(* IEC 61131-3 sources: festo-codesys-mcp/knowledge/library/sensors, 4 files *)

(* ---- FB_AnalogInput.st ---- *)
(* =============================================================
   FB_AnalogInput — Generic Analog Input with Scaling and Filtering

   Category:     Sensors
   Platform:     CODESYS V3.5 (IEC 61131-3)
   Version:      1.0
   Dependencies: None (standard IEC only)

   General-purpose analog input block with linear scaling from
   raw ADC to engineering units, first-order filtering, and
   high/low alarm limits.

   Usage:
     fbPressure : FB_AnalogInput;
     fbPressure(nRawValue := nAD_Ch1,
                rScaleMin := 0.0, rScaleMax := 10.0,
                sUnit := 'bar');
     rPressure := fbPressure.rValue;
   ============================================================= *)
FUNCTION_BLOCK FB_AnalogInput
VAR_INPUT
    nRawValue       : INT;                 (* Raw ADC value *)
    rScaleMin       : REAL := 0.0;         (* Engineering minimum *)
    rScaleMax       : REAL := 100.0;       (* Engineering maximum *)
    nRawMin         : INT := 0;            (* ADC raw minimum *)
    nRawMax         : INT := 32767;        (* ADC raw maximum *)
    rAlarmHigh      : REAL := 90.0;        (* High alarm limit *)
    rAlarmLow       : REAL := 5.0;         (* Low alarm limit *)
    rHysteresis     : REAL := 2.0;         (* Alarm hysteresis *)
    rFilterFactor   : REAL := 0.2;         (* Filter alpha (0.0-1.0) *)
    bEnable         : BOOL := TRUE;        (* Enable processing *)
END_VAR
VAR_OUTPUT
    rValue          : REAL;                (* Scaled value *)
    rPercent        : REAL;                (* 0-100% of scale *)
    bAlarmHigh      : BOOL;                (* High alarm *)
    bAlarmLow       : BOOL;                (* Low alarm *)
    bValid          : BOOL;                (* Reading valid *)
END_VAR
VAR
    rFiltered       : REAL;
    rRange          : REAL;
    bInit           : BOOL := FALSE;
END_VAR

IF NOT bEnable THEN
    bValid := FALSE;
    RETURN;
END_IF

(* Filter *)
IF NOT bInit THEN
    rFiltered := INT_TO_REAL(nRawValue);
    bInit := TRUE;
ELSE
    rFiltered := rFiltered + rFilterFactor * (INT_TO_REAL(nRawValue) - rFiltered);
END_IF

(* Scale *)
rRange := INT_TO_REAL(nRawMax - nRawMin);
IF ABS(rRange) > 0.001 THEN
    rValue := (rFiltered - INT_TO_REAL(nRawMin)) / rRange
              * (rScaleMax - rScaleMin) + rScaleMin;
    rPercent := (rFiltered - INT_TO_REAL(nRawMin)) / rRange * 100.0;
ELSE
    rValue := rScaleMin;
    rPercent := 0.0;
END_IF
bValid := TRUE;

(* Alarms with hysteresis *)
IF rValue >= rAlarmHigh THEN
    bAlarmHigh := TRUE;
ELSIF rValue < (rAlarmHigh - rHysteresis) THEN
    bAlarmHigh := FALSE;
END_IF

IF rValue <= rAlarmLow THEN
    bAlarmLow := TRUE;
ELSIF rValue > (rAlarmLow + rHysteresis) THEN
    bAlarmLow := FALSE;
END_IF

END_FUNCTION_BLOCK

(* ---- FB_FlowSensor.st ---- *)
(* =============================================================
   FB_FlowSensor — Flow Rate Sensor with Totalization

   Category:     Sensors
   Platform:     CODESYS V3.5 (IEC 61131-3)
   Version:      1.0
   Dependencies: None (standard IEC only)

   Monitors flow rate from analog sensor (4-20mA/0-10V).
   Includes low-flow alarm, totalization (accumulated volume),
   and peak flow tracking.

   Usage:
     fbFlow : FB_FlowSensor;
     fbFlow(nRawValue := nAD_Flow,
            rScaleMin := 0.0, rScaleMax := 50.0,
            rAlarmLow := 5.0, tCycleTime := T#100MS);
     rFlowRate  := fbFlow.rValue;
     rTotalVol  := fbFlow.rTotalVolume;
     bNoFlow    := fbFlow.bAlarmLow;
   ============================================================= *)
FUNCTION_BLOCK FB_FlowSensor
VAR_INPUT
    nRawValue       : INT;                 (* Raw ADC value *)
    rScaleMin       : REAL := 0.0;         (* Flow min [L/min] *)
    rScaleMax       : REAL := 50.0;        (* Flow max [L/min] *)
    nRawMin         : INT := 0;            (* ADC minimum *)
    nRawMax         : INT := 32767;        (* ADC maximum *)
    rAlarmLow       : REAL := 5.0;         (* Low flow alarm [L/min] *)
    rHysteresis     : REAL := 1.0;         (* Alarm hysteresis *)
    rFilterFactor   : REAL := 0.15;        (* Filter alpha *)
    tCycleTime      : TIME := T#100MS;     (* PLC scan cycle *)
    bEnable         : BOOL := TRUE;        (* Enable sensor *)
    bResetTotal     : BOOL;                (* Reset totalizer *)
END_VAR
VAR_OUTPUT
    rValue          : REAL;                (* Flow rate [L/min] *)
    rTotalVolume    : REAL := 0.0;         (* Accumulated volume [L] *)
    rPeakFlow       : REAL := 0.0;         (* Peak flow recorded *)
    bAlarmLow       : BOOL;                (* Low flow alarm *)
    bNoFlow         : BOOL;                (* Zero flow detected *)
    bValid          : BOOL;                (* Reading valid *)
END_VAR
VAR
    rFiltered       : REAL;
    rRange          : REAL;
    rDtMin          : REAL;
    bInit           : BOOL := FALSE;
END_VAR

IF bResetTotal THEN
    rTotalVolume := 0.0;
    rPeakFlow := 0.0;
END_IF

IF NOT bEnable THEN
    bValid := FALSE;
    RETURN;
END_IF

(* Filter *)
IF NOT bInit THEN
    rFiltered := INT_TO_REAL(nRawValue);
    bInit := TRUE;
ELSE
    rFiltered := rFiltered + rFilterFactor * (INT_TO_REAL(nRawValue) - rFiltered);
END_IF

(* Scale *)
rRange := INT_TO_REAL(nRawMax - nRawMin);
IF ABS(rRange) > 0.001 THEN
    rValue := (rFiltered - INT_TO_REAL(nRawMin)) / rRange
              * (rScaleMax - rScaleMin) + rScaleMin;
ELSE
    rValue := 0.0;
END_IF
IF rValue < 0.0 THEN rValue := 0.0; END_IF
bValid := TRUE;

(* Totalization: flow [L/min] * dt [min] = volume [L] *)
rDtMin := TIME_TO_REAL(tCycleTime) / 60000.0;  (* ms → minutes *)
rTotalVolume := rTotalVolume + rValue * rDtMin;

(* Peak tracking *)
IF rValue > rPeakFlow THEN
    rPeakFlow := rValue;
END_IF

(* Alarms *)
bNoFlow := rValue < 0.5;
IF rValue <= rAlarmLow THEN bAlarmLow := TRUE;
ELSIF rValue > (rAlarmLow + rHysteresis) THEN bAlarmLow := FALSE; END_IF

END_FUNCTION_BLOCK

(* ---- FB_LevelSensor.st ---- *)
(* =============================================================
   FB_LevelSensor — Tank Level Sensor with Alarms

   Category:     Sensors
   Platform:     CODESYS V3.5 (IEC 61131-3)
   Version:      1.0
   Dependencies: None (standard IEC only)

   Monitors liquid level in tanks/reservoirs. Supports continuous
   analog input (4-20mA/0-10V) with high/low alarms and
   optional float switch inputs for redundant level detection.

   Usage:
     fbLevel : FB_LevelSensor;
     fbLevel(nRawValue := nAD_Level,
             rScaleMin := 0.0, rScaleMax := 100.0,
             rAlarmHigh := 95.0, rAlarmLow := 10.0,
             bFloatHigh := bDI_FloatHigh,
             bFloatLow := bDI_FloatLow);
     rLevelPercent := fbLevel.rValue;
     bRefillNeeded := fbLevel.bAlarmLow;
   ============================================================= *)
FUNCTION_BLOCK FB_LevelSensor
VAR_INPUT
    nRawValue       : INT;                 (* Raw ADC value *)
    rScaleMin       : REAL := 0.0;         (* Level minimum [%] *)
    rScaleMax       : REAL := 100.0;       (* Level maximum [%] *)
    nRawMin         : INT := 0;            (* ADC minimum *)
    nRawMax         : INT := 32767;        (* ADC maximum *)
    rAlarmHigh      : REAL := 95.0;        (* High level alarm [%] *)
    rAlarmLow       : REAL := 10.0;        (* Low level alarm [%] *)
    rWarnLow        : REAL := 20.0;        (* Low level warning [%] *)
    rHysteresis     : REAL := 3.0;         (* Alarm hysteresis *)
    rFilterFactor   : REAL := 0.05;        (* Filter (slow for level) *)
    bFloatHigh      : BOOL := FALSE;       (* Float switch: high level *)
    bFloatLow       : BOOL := TRUE;        (* Float switch: low level (NC) *)
    bUseFloats      : BOOL := FALSE;       (* Use float switches for alarms *)
    bEnable         : BOOL := TRUE;        (* Enable sensor *)
END_VAR
VAR_OUTPUT
    rValue          : REAL;                (* Level [%] *)
    bAlarmHigh      : BOOL;                (* High level alarm *)
    bAlarmLow       : BOOL;                (* Low level alarm *)
    bWarnLow        : BOOL;                (* Low level warning *)
    bEmpty          : BOOL;                (* Tank empty *)
    bFull           : BOOL;                (* Tank full *)
    bValid          : BOOL;                (* Reading valid *)
END_VAR
VAR
    rFiltered       : REAL;
    rRange          : REAL;
    bInit           : BOOL := FALSE;
END_VAR

IF NOT bEnable THEN
    bValid := FALSE;
    RETURN;
END_IF

(* Filter *)
IF NOT bInit THEN
    rFiltered := INT_TO_REAL(nRawValue);
    bInit := TRUE;
ELSE
    rFiltered := rFiltered + rFilterFactor * (INT_TO_REAL(nRawValue) - rFiltered);
END_IF

(* Scale *)
rRange := INT_TO_REAL(nRawMax - nRawMin);
IF ABS(rRange) > 0.001 THEN
    rValue := (rFiltered - INT_TO_REAL(nRawMin)) / rRange
              * (rScaleMax - rScaleMin) + rScaleMin;
ELSE
    rValue := rScaleMin;
END_IF

(* Clamp *)
IF rValue > rScaleMax THEN rValue := rScaleMax; END_IF
IF rValue < rScaleMin THEN rValue := rScaleMin; END_IF
bValid := TRUE;

(* Alarms — analog or float switch based *)
IF bUseFloats THEN
    bAlarmHigh := bFloatHigh;
    bAlarmLow  := NOT bFloatLow;  (* NC float: open = low level *)
ELSE
    IF rValue >= rAlarmHigh THEN bAlarmHigh := TRUE;
    ELSIF rValue < (rAlarmHigh - rHysteresis) THEN bAlarmHigh := FALSE; END_IF

    IF rValue <= rAlarmLow THEN bAlarmLow := TRUE;
    ELSIF rValue > (rAlarmLow + rHysteresis) THEN bAlarmLow := FALSE; END_IF
END_IF

(* Warning *)
IF rValue <= rWarnLow THEN bWarnLow := TRUE;
ELSIF rValue > (rWarnLow + rHysteresis) THEN bWarnLow := FALSE; END_IF

bEmpty := rValue <= rScaleMin + 1.0;
bFull  := rValue >= rScaleMax - 1.0;

END_FUNCTION_BLOCK

(* ---- FB_TemperatureSensor.st ---- *)
(* =============================================================
   FB_TemperatureSensor — Universal Temperature Sensor Interface

   Category:     Sensors
   Platform:     CODESYS V3.5 (IEC 61131-3)
   Version:      1.0
   Dependencies: None (standard IEC only)

   Supports three input types:
   - 4-20mA transmitter (nInputType := 0)
   - 0-10V transmitter  (nInputType := 1)
   - Direct PT100 RTD   (nInputType := 2)

   Features: scaling, wire-break/short detection, high/low alarms
   with hysteresis, first-order filter.

   Usage:
     fbTemp : FB_TemperatureSensor;
     fbTemp(nRawValue := nAD_Ch0, nInputType := 0,
            rScaleMin := 0.0, rScaleMax := 200.0,
            rAlarmHigh := 180.0, rAlarmLow := 5.0);
     rTemperature := fbTemp.rValue;
     bOverTemp    := fbTemp.bAlarmHigh;
   ============================================================= *)
FUNCTION_BLOCK FB_TemperatureSensor
VAR_INPUT
    nRawValue       : INT;                 (* Raw ADC value *)
    nInputType      : INT := 0;            (* 0=4-20mA, 1=0-10V, 2=PT100 *)
    rScaleMin       : REAL := 0.0;         (* Eng. unit at raw min [deg C] *)
    rScaleMax       : REAL := 200.0;       (* Eng. unit at raw max [deg C] *)
    nRawMin         : INT := 0;            (* Raw ADC minimum *)
    nRawMax         : INT := 32767;        (* Raw ADC maximum *)
    rAlarmHigh      : REAL := 180.0;       (* High alarm threshold *)
    rAlarmLow       : REAL := 5.0;         (* Low alarm threshold *)
    rWarnHigh       : REAL := 150.0;       (* High warning threshold *)
    rWarnLow        : REAL := 10.0;        (* Low warning threshold *)
    rHysteresis     : REAL := 2.0;         (* Alarm hysteresis *)
    rFilterFactor   : REAL := 0.1;         (* Low-pass filter (0.0-1.0) *)
    nWireBreakLow   : INT := 100;          (* Wire break detection: below this = open *)
    nWireBreakHigh  : INT := 32600;        (* Wire break detection: above this = short *)
    bEnable         : BOOL := TRUE;        (* Enable sensor processing *)
END_VAR
VAR_OUTPUT
    rValue          : REAL;                (* Scaled temperature [deg C] *)
    rRawFiltered    : REAL;                (* Filtered raw value *)
    bAlarmHigh      : BOOL;                (* High alarm active *)
    bAlarmLow       : BOOL;               (* Low alarm active *)
    bWarnHigh       : BOOL;                (* High warning active *)
    bWarnLow        : BOOL;                (* Low warning active *)
    bWireBreak      : BOOL;                (* Wire break / open circuit *)
    bShortCircuit   : BOOL;                (* Short circuit detected *)
    bErr          : BOOL;                (* Any error condition *)
    bValid          : BOOL;                (* Reading is valid *)
END_VAR
VAR
    rRawReal        : REAL;
    rScaled         : REAL;
    rRange          : REAL;
    bInit           : BOOL := FALSE;
END_VAR

IF NOT bEnable THEN
    bValid := FALSE;
    RETURN;
END_IF

rRawReal := INT_TO_REAL(nRawValue);

(* Wire break / short circuit detection *)
bWireBreak    := nRawValue < nWireBreakLow;
bShortCircuit := nRawValue > nWireBreakHigh;
bErr        := bWireBreak OR bShortCircuit;

IF bErr THEN
    bValid := FALSE;
    RETURN;
END_IF

(* First-order low-pass filter *)
IF NOT bInit THEN
    rRawFiltered := rRawReal;
    bInit := TRUE;
ELSE
    rRawFiltered := rRawFiltered + rFilterFactor * (rRawReal - rRawFiltered);
END_IF

(* Linear scaling: raw → engineering units *)
rRange := INT_TO_REAL(nRawMax - nRawMin);
IF ABS(rRange) > 0.001 THEN
    rScaled := (rRawFiltered - INT_TO_REAL(nRawMin)) / rRange
               * (rScaleMax - rScaleMin) + rScaleMin;
ELSE
    rScaled := rScaleMin;
END_IF
rValue := rScaled;
bValid := TRUE;

(* Alarm evaluation with hysteresis *)
IF rValue >= rAlarmHigh THEN
    bAlarmHigh := TRUE;
ELSIF rValue < (rAlarmHigh - rHysteresis) THEN
    bAlarmHigh := FALSE;
END_IF

IF rValue <= rAlarmLow THEN
    bAlarmLow := TRUE;
ELSIF rValue > (rAlarmLow + rHysteresis) THEN
    bAlarmLow := FALSE;
END_IF

IF rValue >= rWarnHigh THEN
    bWarnHigh := TRUE;
ELSIF rValue < (rWarnHigh - rHysteresis) THEN
    bWarnHigh := FALSE;
END_IF

IF rValue <= rWarnLow THEN
    bWarnLow := TRUE;
ELSIF rValue > (rWarnLow + rHysteresis) THEN
    bWarnLow := FALSE;
END_IF

END_FUNCTION_BLOCK
